(* IEC 61131-3 sources: volt/packages/volt-lsp-iec/test-corpus/pro2193/Device/Plc Logic/Application/03 Hardware Units/31 SER/31.22 - Reject Stations/With blowoff, 1 file *)

(* ---- RejectStation_WithBlowOffFB.pou ---- *)
{attribute 'symbol' := 'none'}
FUNCTION_BLOCK RejectStation_WithBlowOffFB
EXTENDS RejectStation_BaseFB
IMPLEMENTS IRejectStation_WithBlowOff_Commands
VAR_INPUT
	{attribute 'symbol' := 'readwrite'}	BlowOff						: ActuatorWithManualControlFB;
END_VAR
VAR_OUTPUT
END_VAR
VAR_IN_OUT
	DataWithBlowOff			: RejectStation_WithBlowOff_Data;
END_VAR
VAR//VISU
END_VAR
VAR
END_VAR

%LANGUAGE ST
SUPER^(Data := Data);

END_FUNCTION_BLOCK

METHOD PROTECTED Cyclic
VAR_INST
	BlowOffDuration						: BTON;
END_VAR

%LANGUAGE ST
SUPER^.Cyclic();

BlowOff(
	manualControlEnabled	:= SER.ManualControlEnabled AND ExternalManualControlEnabled);

DataWithBlowOff.rBlowOffDuration	:= LIMIT(0.05, DataWithBlowOff.rBlowOffDuration, 5);

IF BlowOffDuration.Set(In := BlowOff.Map(), Pt := DataWithBlowOff.rBlowOffDuration) THEN
	BlowOff.Reset();
END_IF

END_METHOD

// Command to reset the module (Statemachine to zero state) in case of E-Stop
METHOD PUBLIC EStop : BOOL	// Returns true when drives are in standstill

%LANGUAGE ST
%FOLDER Commands
BlowOff.Reset();

EStop := SUPER^.EStop();

END_METHOD

// Receive a certain amount of products by vacuum or clamps. Parameter indicates which product is received.
METHOD PUBLIC GetProducts : BOOL
VAR_INPUT
	vacuumIndex		: WORD;	// 0: All vacuums, bit 1: Vacuum 1, bit 2: Vacuum 2, etc.
END_VAR

%LANGUAGE ST
%FOLDER Commands
IF NOT CommandLock.Request(__POUNAME()) THEN
	RETURN;
END_IF

IF CommandLock.FirstCall THEN
	BlowOff.Set();
END_IF

//IF NOT BlowOff.Map() THEN
	GetProducts := CommandLock.Release(__POUNAME());
//END_IF

END_METHOD

// Command to reset the module. Servodrives are homed.
METHOD PUBLIC Reset : BOOL	// Returns true when homing done

%LANGUAGE ST
%FOLDER Commands
BlowOff.Reset();

Reset := SUPER^.Reset();

END_METHOD

// Command to reset the module (Statemachine to zero state)
METHOD PUBLIC Stop : BOOL	// Returns true when drives are in standstill

%LANGUAGE ST
%FOLDER Commands
BlowOff.Reset();

Stop := SUPER^.Stop();

END_METHOD
